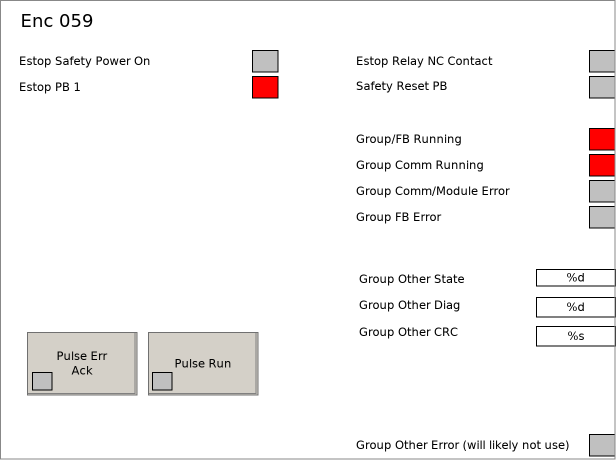
VISUALIZATION SafetyConv_Enc059  // 616x460
    Rectangle (252,50 26x22), colour toggle: SafetyInterface_Enc059.fbSafetyInterface.hoSafetyPowerOn_Estop
    Rectangle (16,46 224x30), "Estop Safety Power On"
    Rectangle (252,76 26x22), colour toggle: SafetyInterface_Enc059.fbSafetyInterface.hoEstopPB1Ok
    Rectangle (16,72 224x30), "Estop PB 1"
    Rectangle (589,50 26x22), colour toggle: SafetyInterface_Enc059.fbSafetyInterface.hoRelayNCContact_Estop
    Rectangle (353,46 224x30), "Estop Relay NC Contact"
    Rectangle (589,128 26x22), colour toggle: SafetyInterface_Enc059.fbSafetyInterface.hoSafetyGroupAndFBInRun
    Rectangle (353,124 224x30), "Group/FB Running"
    Rectangle (589,154 26x22), colour toggle: SafetyInterface_Enc059.fbSafetyInterface.hoSafetyGroupComRunning
    Rectangle (353,150 224x30), "Group Comm Running"
    Rectangle (589,180 26x22), colour toggle: SafetyInterface_Enc059.fbSafetyInterface.hoSafetyGroupComErr
    Rectangle (353,176 224x30), "Group Comm/Module Error"
    Rectangle (589,206 26x22), colour toggle: SafetyInterface_Enc059.fbSafetyInterface.hoSafetyGroupFBErr
    Rectangle (353,202 224x30), "Group FB Error"
    Rectangle (589,434 26x22), colour toggle: SafetyInterface_Enc059.fbSafetyInterface.hoSafetyGroupOtherErr
    Rectangle (353,430 224x30), "Group Other Error (will likely not use)"
    Rectangle (356,264 224x30), "Group Other State"
    Rectangle (356,290 224x30), "Group Other Diag"
    Rectangle (536,269 80x17), "%d", text variable: SafetyInterface_Enc059.fbSafetyInterface.hoSafetyGroup_State
    Rectangle (536,297 80x20), "%d", text variable: SafetyInterface_Enc059.fbSafetyInterface.hoSafetyGroup_Diag
    Button (27,332 110x63), "Pulse Err Ack"
        tap SafetyInterface_Enc059.fbSafetyInterface.hiSafetyGroupPulseErrAck
    Button (148,332 110x63), "Pulse Run"
        tap SafetyInterface_Enc059.fbSafetyInterface.hiSafetyGroupPulseRun
    Rectangle (152,372 20x18), colour toggle: SafetyInterface_Enc059.fbSafetyInterface.hoSafetyGroupRun
    Rectangle (32,372 20x18), colour toggle: SafetyInterface_Enc059.fbSafetyInterface.hoSafetyGroupErrAck
    Rectangle (356,317 224x30), "Group Other CRC"
    RoundedRectangle (536,326 80x20), "%s", text variable: SafetyInterface_Enc059.fbSafetyInterface.hoSafetyCtrlCRC, colour variable: 16#FF000000 OR (16#FF000000 OR (Global_Variables.gStn100.OperatorMessage.Color))
    Rectangle (589,76 26x22), colour toggle: SafetyInterface_Enc059.fbSafetyInterface.hoSafetyResetPB
    Rectangle (353,71 224x30), "Safety Reset PB"
    Label (16,12 82x18), "Enc 059"
END_VISUALIZATION

(* stored: Version 1.1.0.1, ProductVersion 3.1.4024.6
   Visu SafetyConv_Enc059: Id {902b6e3e-0ad3-4291-9043-d725d990afbc} *)
